# EPICS substitutions: snmpApp/Db/snmp_ping.substitutions
file snmp_mbbi.template {
pattern
{        P,       ATTR,                   DESC,                                                OID,        SCAN,      ZRST, ONST,   TWST,     ZRSV,     ONSV,     TWSV}
{   SPEAR1, PingStatus,   "SPEAR1 ping status", .1.3.6.1.4.1.8072.1.3.2.3.1.4.5.112.105.110.103.49, "10 second", "Unknown", "Up", "Down",    MAJOR, NO_ALARM,    MAJOR}
{   SPEAR2, PingStatus,   "SPEAR2 ping status", .1.3.6.1.4.1.8072.1.3.2.3.1.4.5.112.105.110.103.50, "10 second", "Unknown", "Up", "Down",    MAJOR, NO_ALARM,    MAJOR}
{    INJ02, PingStatus,    "INJ02 ping status", .1.3.6.1.4.1.8072.1.3.2.3.1.4.5.112.105.110.103.51, "10 second", "Unknown", "Up", "Down",    MAJOR, NO_ALARM,    MAJOR}
{ SPEARNFS, PingStatus, "SPEARNFS ping status", .1.3.6.1.4.1.8072.1.3.2.3.1.4.5.112.105.110.103.52, "10 second", "Unknown", "Up", "Down",    MAJOR, NO_ALARM,    MAJOR}
}
